(* Simple binary user data (8 byte aligned) *)
TYPE ST_ApplicationBinaryData :
STRUCT
	fPos		:  LREAL;(* 8 byte *)
END_STRUCT
END_TYPE

(* stored: Version 1.1.0.1, ProductVersion 3.1.4024.12
   DUT ST_ApplicationBinaryData: Id {1d93b951-d881-4acd-a086-da3415ea1d6d} *)
